KUKA KRL program: Gripper_check.src, Gripper_check.dat

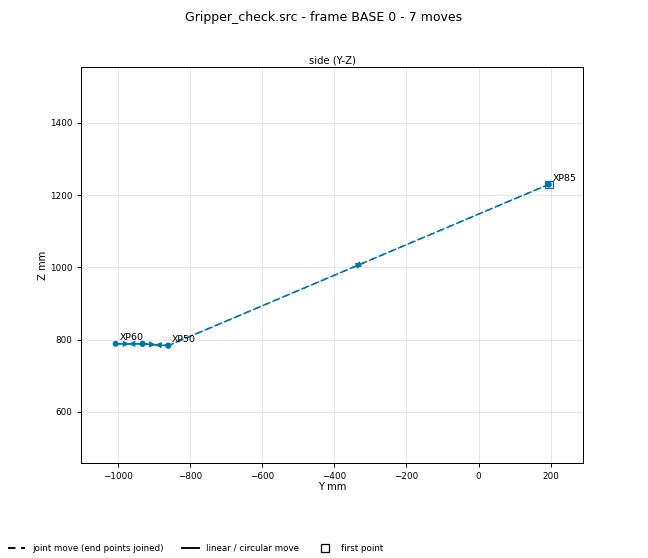
[picture p0: tool path of Gripper_check.src in frame BASE 0, 7 of 9 moves have a stored position in this frame; points joined in program order, loops and branches not executed]
--- Gripper_check.src ---
&ACCESS RVP
&REL 175
&PARAM EDITMASK = *
&PARAM TEMPLATE = C:\KRC\Roboter\Template\vorgabe
&PARAM DISKPATH = KRC:\R1\Program\Sevice Programs
DEF Gripper_check( )
;FOLD INI;%{PE}
  ;FOLD BASISTECH INI
    GLOBAL INTERRUPT DECL 3 WHEN $STOPMESS==TRUE DO IR_STOPM ( )
    INTERRUPT ON 3
    BAS (#INITMOV,0 )
  ;ENDFOLD (BASISTECH INI)
;FOLD SPOTTECH INI
USERSPOT(#INIT)
;ENDFOLD (SPOTTECH INI)
;FOLD GRIPPERTECH INI
USER_GRP(0,DUMMY,DUMMY,GDEFAULT)
;ENDFOLD (GRIPPERTECH INI)
  ;FOLD USER INI
    ;Make your modifications here

  ;ENDFOLD (USER INI)
;ENDFOLD (INI)

;FOLD PTP HOME  Vel= 100 % DEFAULT;%{PE}%MKUKATPBASIS,%CMOVE,%VPTP,%P 1:PTP, 2:HOME, 3:, 5:100, 7:DEFAULT
$BWDSTART = FALSE
PDAT_ACT=PDEFAULT
FDAT_ACT=FHOME
BAS (#PTP_PARAMS,100 )
$H_POS=XHOME
PTP  XHOME
;ENDFOLD

;FOLD PTP P85 Vel=100 % H Tool[5] Base[0];%{PE}%R 8.3.48,%MKUKATPBASIS,%CMOVE,%VPTP,%P 1:PTP, 2:P85, 3:, 5:100, 7:H
$BWDSTART=FALSE
PDAT_ACT=PH
FDAT_ACT=FP85
BAS(#PTP_PARAMS,100)
PTP XP85
;ENDFOLD
;FOLD PTP P50 Vel=100 % H Tool[5] Base[0];%{PE}%R 8.3.48,%MKUKATPBASIS,%CMOVE,%VPTP,%P 1:PTP, 2:P50, 3:, 5:100, 7:H
$BWDSTART=FALSE
PDAT_ACT=PH
FDAT_ACT=FP50
BAS(#PTP_PARAMS,100)
PTP XP50
;ENDFOLD

;FOLD WAIT FOR ( IN 246 'Grps: bat reposo' ) CONT;%{PE}%R 8.3.48 %MKUKATPBASIS %CEXT_WAIT_FOR %VEXT_WAIT_FOR,%P 2:, 4:, 5:$IN, 6:246, 7:Grps: bat reposo, 9:CONTINUE
CONTINUE
WAIT FOR  ( $IN[246] )
;ENDFOLD
;FOLD WAIT FOR ( IN 248 'Grps: bat reposo' ) CONT;%{PE}%R 8.3.48 %MKUKATPBASIS %CEXT_WAIT_FOR %VEXT_WAIT_FOR,%P 2:, 4:, 5:$IN, 6:248, 7:Grps: bat reposo, 9:CONTINUE
CONTINUE
WAIT FOR  ( $IN[248] )
;ENDFOLD

;FOLD LIN P52 Vel=0.1 m/s M Tool[5] Base[0];%{PE}%R 8.3.48,%MKUKATPBASIS,%CMOVE,%VLIN,%P 1:LIN, 2:P52, 3:, 5:0.1, 7:M
$BWDSTART=FALSE
LDAT_ACT=LM
FDAT_ACT=FP52
BAS(#CP_PARAMS,0.1)
LIN XP52
;ENDFOLD

;Pos Galga
;FOLD LIN P60 Vel=0.01 m/s L Tool[5] Base[0];%{PE}%R 8.3.48,%MKUKATPBASIS,%CMOVE,%VLIN,%P 1:LIN, 2:P60, 3:, 5:0.01, 7:L
$BWDSTART=FALSE
LDAT_ACT=LL
FDAT_ACT=FP60
BAS(#CP_PARAMS,0.01)
LIN XP60
;ENDFOLD
HALT

;Cierra pinchos
;FOLD OUT 243 'cil bat reposo' State=FALSE ;%{PE}%R 8.3.48,%MKUKATPBASIS,%COUT,%VOUTX,%P 2:243, 3:cil bat reposo, 5:FALSE, 6:
$OUT[243]=FALSE
;ENDFOLD
;FOLD OUT 244 'cil bat activo' State=TRUE ;%{PE}%R 8.3.48,%MKUKATPBASIS,%COUT,%VOUTX,%P 2:244, 3:cil bat activo, 5:TRUE, 6:
$OUT[244]=TRUE
;ENDFOLD
;FOLD WAIT FOR ( IN 245 'Grps: bat activo' );%{PE}%R 8.3.48 %MKUKATPBASIS %CEXT_WAIT_FOR %VEXT_WAIT_FOR,%P 2:, 4:, 5:$IN, 6:245, 7:Grps: bat activo, 9:
WAIT FOR  ( $IN[245] )
;ENDFOLD
;FOLD WAIT FOR ( IN 247 'Grps: baterias activo' );%{PE}%R 8.3.48 %MKUKATPBASIS %CEXT_WAIT_FOR %VEXT_WAIT_FOR,%P 2:, 4:, 5:$IN, 6:247, 7:Grps: baterias activo, 9:
WAIT FOR  ( $IN[247] )
;ENDFOLD
HALT

;aBRE pinchos
;FOLD OUT 244 'cil bat activo' State=FALSE ;%{PE}%R 8.3.48,%MKUKATPBASIS,%COUT,%VOUTX,%P 2:244, 3:cil bat activo, 5:FALSE, 6:
$OUT[244]=FALSE
;ENDFOLD
;FOLD OUT 243 'cil bat reposo' State=TRUE ;%{PE}%R 8.3.48,%MKUKATPBASIS,%COUT,%VOUTX,%P 2:243, 3:cil bat reposo, 5:TRUE, 6:
$OUT[243]=TRUE
;ENDFOLD
;FOLD WAIT FOR ( IN 246 'Grps: bat reposo' AND IN 248 'Grps: bat reposo' );%{PE}%R 8.3.48 %MKUKATPBASIS %CEXT_WAIT_FOR %VEXT_WAIT_FOR,%P 2:, 4:, 5:$IN, 6:246, 7:Grps: bat reposo, 8:AND, 9:, 10:$IN, 11:248, 12:Grps: bat reposo, 14:
WAIT FOR  ( $IN[246] AND $IN[248] )
;ENDFOLD
;FOLD WAIT Time=1 sec;%{PE}%R 8.3.48,%MKUKATPBASIS,%CWAIT,%VWAIT,%P 3:1
WAIT SEC 1
;ENDFOLD

;Retirada
;FOLD LIN P55 CONT Vel=2 m/s M Tool[5] Base[0];%{PE}%R 8.3.48,%MKUKATPBASIS,%CMOVE,%VLIN,%P 1:LIN, 2:P55, 3:C_DIS C_DIS, 5:2, 7:M
$BWDSTART=FALSE
LDAT_ACT=LM
FDAT_ACT=FP55
BAS(#CP_PARAMS,2)
LIN XP55 C_DIS C_DIS
;ENDFOLD
;FOLD PTP P54 Vel=100 % H Tool[5] Base[0];%{PE}%R 8.3.48,%MKUKATPBASIS,%CMOVE,%VPTP,%P 1:PTP, 2:P54, 3:, 5:100, 7:H
$BWDSTART=FALSE
PDAT_ACT=PH
FDAT_ACT=FP54
BAS(#PTP_PARAMS,100)
PTP XP54
;ENDFOLD
;FOLD PTP P53 Vel=100 % H Tool[5] Base[0];%{PE}%R 8.3.48,%MKUKATPBASIS,%CMOVE,%VPTP,%P 1:PTP, 2:P53, 3:, 5:100, 7:H
$BWDSTART=FALSE
PDAT_ACT=PH
FDAT_ACT=FP53
BAS(#PTP_PARAMS,100)
PTP XP53
;ENDFOLD
HALT

;FOLD PTP HOME  Vel= 100 % DEFAULT;%{PE}%MKUKATPBASIS,%CMOVE,%VPTP,%P 1:PTP, 2:HOME, 3:, 5:100, 7:DEFAULT
$BWDSTART = FALSE
PDAT_ACT=PDEFAULT
FDAT_ACT=FHOME
BAS (#PTP_PARAMS,100 )
$H_POS=XHOME
PTP  XHOME
;ENDFOLD
END

--- Gripper_check.dat ---
&ACCESS RVP
&REL 175
&PARAM EDITMASK = *
&PARAM TEMPLATE = C:\KRC\Roboter\Template\vorgabe
&PARAM DISKPATH = KRC:\R1\Program\Sevice Programs
DEFDAT  Gripper_check
;FOLD EXTERNAL DECLARATIONS;%{PE}%MKUKATPBASIS,%CEXT,%VCOMMON,%P
;FOLD GRIPPERTECH EXT
EXT  H50 (INT  :IN,INT  :IN,INT  :IN,GRP_TYP  :IN )
;ENDFOLD (GRIPPERTECH EXT)
;FOLD SPOTTECH EXT
EXT  USERSPOT (S_COMMAND  :IN,SPOT_TYPE  :IN )
;ENDFOLD (SPOTTECH EXT)
;FOLD BASISTECH EXT;%{PE}%MKUKATPBASIS,%CEXT,%VEXT,%P
EXT  BAS (BAS_COMMAND  :IN,REAL  :IN )
DECL INT SUCCESS
;ENDFOLD (BASISTECH EXT)
;FOLD USER EXT;%{E}%MKUKATPUSER,%CEXT,%VEXT,%P
;Make your modifications here

;ENDFOLD (USER EXT)
;ENDFOLD (EXTERNAL DECLARATIONS)
DECL BASIS_SUGG_T LAST_BASIS={POINT1[] "P60b                    ",POINT2[] "P60b                    ",CP_PARAMS[] "M                       ",PTP_PARAMS[] "H                       ",CONT[] "                        ",CP_VEL[] "2                       ",PTP_VEL[] "100                     ",SYNC_PARAMS[] "SYNCDAT                 ",SPL_NAME[] "S0                      ",A_PARAMS[] "ADAT0                   "}
DECL E6POS XP50={X 952.374695,Y -860.111694,Z 783.046143,A 80.5366592,B 88.5556259,C 169.570068,S 6,T 26,E1 0.0,E2 0.0,E3 0.0,E4 0.0,E5 0.0,E6 0.0}
DECL FDAT FP50={TOOL_NO 5,BASE_NO 0,IPO_FRAME #BASE,POINT2[] " ",TQ_STATE FALSE}
DECL PDAT PH={VEL 100.000,ACC 100.000,APO_DIST 100.000,APO_MODE #CDIS,GEAR_JERK 50.0000,EXAX_IGN 0}
DECL E6POS XP60={X 952.955505,Y -1005.88715,Z 788.139,A 20.0385742,B 89.1085663,C 109.304688,S 6,T 26,E1 0.0,E2 0.0,E3 0.0,E4 0.0,E5 0.0,E6 0.0}
DECL FDAT FP60={TOOL_NO 5,BASE_NO 0,IPO_FRAME #BASE,POINT2[] " ",TQ_STATE FALSE}
DECL LDAT LL={VEL 2.00000,ACC 25.0000,APO_DIST 100.000,APO_FAC 50.0000,AXIS_VEL 100.000,AXIS_ACC 100.000,ORI_TYP #VAR,CIRC_TYP #BASE,JERK_FAC 50.0000,GEAR_JERK 50.0000,EXAX_IGN 0}
DECL E6POS XP51={X 1024.76611,Y -1067.43542,Z 519.066956,A 55.3303528,B 87.7738342,C 145.849503,S 6,T 26,E1 0.0,E2 0.0,E3 0.0,E4 0.0,E5 0.0,E6 0.0}
DECL FDAT FP51={TOOL_NO 5,BASE_NO 0,IPO_FRAME #BASE,POINT2[] " ",TQ_STATE FALSE}
DECL E6POS XP70={X 1027.60229,Y -977.170227,Z 520.707,A 88.3586,B 88.2946472,C 177.924576,S 6,T 26,E1 0.0,E2 0.0,E3 0.0,E4 0.0,E5 0.0,E6 0.0}
DECL FDAT FP70={TOOL_NO 5,BASE_NO 0,IPO_FRAME #BASE,POINT2[] " ",TQ_STATE FALSE}
DECL E6POS XP52={X 952.798523,Y -931.386414,Z 788.051941,A 20.3578415,B 89.1093369,C 109.624481,S 6,T 26,E1 0.0,E2 0.0,E3 0.0,E4 0.0,E5 0.0,E6 0.0}
DECL FDAT FP52={TOOL_NO 5,BASE_NO 0,IPO_FRAME #BASE,POINT2[] " ",TQ_STATE FALSE}
DECL LDAT LM={VEL 2.00000,ACC 25.0000,APO_DIST 100.000,APO_FAC 50.0000,AXIS_VEL 100.000,AXIS_ACC 100.000,ORI_TYP #VAR,CIRC_TYP #BASE,JERK_FAC 50.0000,GEAR_JERK 50.0000,EXAX_IGN 0}
DECL E6POS XP53={X 938.561218,Y 193.717773,Z 1229.66455,A 174.754501,B 24.9198875,C -153.479370,S 6,T 27,E1 0.0,E2 0.0,E3 0.0,E4 0.0,E5 0.0,E6 0.0}
DECL FDAT FP53={TOOL_NO 5,BASE_NO 0,IPO_FRAME #BASE,POINT2[] " ",TQ_STATE FALSE}
DECL E6POS XP54={X 952.374695,Y -860.111694,Z 783.046143,A 80.5366592,B 88.5556259,C 169.570068,S 6,T 26,E1 0.0,E2 0.0,E3 0.0,E4 0.0,E5 0.0,E6 0.0}
DECL FDAT FP54={TOOL_NO 5,BASE_NO 0,IPO_FRAME #BASE,POINT2[] " ",TQ_STATE FALSE}
DECL E6POS XP55={X 952.798523,Y -931.386414,Z 788.051941,A 20.3578415,B 89.1093369,C 109.624481,S 6,T 26,E1 0.0,E2 0.0,E3 0.0,E4 0.0,E5 0.0,E6 0.0}
DECL FDAT FP55={TOOL_NO 5,BASE_NO 0,IPO_FRAME #BASE,POINT2[] " ",TQ_STATE FALSE}
DECL E6POS XP56={X 1023.94318,Y -901.988892,Z 779.185486,A 84.6670,B 88.5756149,C 177.274,S 6,T 26,E1 0.0,E2 0.0,E3 0.0,E4 0.0,E5 0.0,E6 0.0}
DECL FDAT FP56={TOOL_NO 5,BASE_NO 0,IPO_FRAME #BASE,POINT2[] " ",TQ_STATE FALSE}
DECL E6POS XP57={X 1023.94318,Y -901.988892,Z 779.185486,A 84.6670,B 88.5756149,C 177.274,S 6,T 26,E1 0.0,E2 0.0,E3 0.0,E4 0.0,E5 0.0,E6 0.0}
DECL FDAT FP57={TOOL_NO 5,BASE_NO 0,IPO_FRAME #BASE,POINT2[] " ",TQ_STATE FALSE}
DECL E6POS XP58={X 1023.94318,Y -901.988892,Z 779.185486,A 84.6670,B 88.5756149,C 177.274,S 6,T 26,E1 0.0,E2 0.0,E3 0.0,E4 0.0,E5 0.0,E6 0.0}
DECL FDAT FP58={TOOL_NO 5,BASE_NO 0,IPO_FRAME #BASE,POINT2[] " ",TQ_STATE FALSE}
DECL E6POS XP59={X 1023.94318,Y -901.988892,Z 779.185486,A 84.6670,B 88.5756149,C 177.274,S 6,T 26,E1 0.0,E2 0.0,E3 0.0,E4 0.0,E5 0.0,E6 0.0}
DECL FDAT FP59={TOOL_NO 5,BASE_NO 0,IPO_FRAME #BASE,POINT2[] " ",TQ_STATE FALSE}
DECL E6POS XP61={X 1023.94318,Y -901.988892,Z 779.185486,A 84.6670,B 88.5756149,C 177.274,S 6,T 26,E1 0.0,E2 0.0,E3 0.0,E4 0.0,E5 0.0,E6 0.0}
DECL FDAT FP61={TOOL_NO 5,BASE_NO 0,IPO_FRAME #BASE,POINT2[] " ",TQ_STATE FALSE}
DECL E6POS XP62={X 1023.94318,Y -901.988892,Z 779.185486,A 84.6670,B 88.5756149,C 177.274,S 6,T 26,E1 0.0,E2 0.0,E3 0.0,E4 0.0,E5 0.0,E6 0.0}
DECL FDAT FP62={TOOL_NO 5,BASE_NO 0,IPO_FRAME #BASE,POINT2[] " ",TQ_STATE FALSE}
DECL E6POS XP63={X 1023.94318,Y -901.988892,Z 779.185486,A 84.6670,B 88.5756149,C 177.274,S 6,T 26,E1 0.0,E2 0.0,E3 0.0,E4 0.0,E5 0.0,E6 0.0}
DECL FDAT FP63={TOOL_NO 5,BASE_NO 0,IPO_FRAME #BASE,POINT2[] " ",TQ_STATE FALSE}
DECL E6POS XP64={X 1023.94318,Y -901.988892,Z 779.185486,A 84.6670,B 88.5756149,C 177.274,S 6,T 26,E1 0.0,E2 0.0,E3 0.0,E4 0.0,E5 0.0,E6 0.0}
DECL FDAT FP64={TOOL_NO 5,BASE_NO 0,IPO_FRAME #BASE,POINT2[] " ",TQ_STATE FALSE}
DECL E6POS XP65={X 1023.94318,Y -901.988892,Z 779.185486,A 84.6670,B 88.5756149,C 177.274,S 6,T 26,E1 0.0,E2 0.0,E3 0.0,E4 0.0,E5 0.0,E6 0.0}
DECL FDAT FP65={TOOL_NO 5,BASE_NO 0,IPO_FRAME #BASE,POINT2[] " ",TQ_STATE FALSE}
DECL E6POS XP66={X 1023.94318,Y -901.988892,Z 779.185486,A 84.6670,B 88.5756149,C 177.274,S 6,T 26,E1 0.0,E2 0.0,E3 0.0,E4 0.0,E5 0.0,E6 0.0}
DECL FDAT FP66={TOOL_NO 5,BASE_NO 0,IPO_FRAME #BASE,POINT2[] " ",TQ_STATE FALSE}
DECL E6POS XP67={X 1023.94318,Y -901.988892,Z 779.185486,A 84.6670,B 88.5756149,C 177.274,S 6,T 26,E1 0.0,E2 0.0,E3 0.0,E4 0.0,E5 0.0,E6 0.0}
DECL FDAT FP67={TOOL_NO 5,BASE_NO 0,IPO_FRAME #BASE,POINT2[] " ",TQ_STATE FALSE}
DECL E6POS XP68={X 1023.94318,Y -901.988892,Z 779.185486,A 84.6670,B 88.5756149,C 177.274,S 6,T 26,E1 0.0,E2 0.0,E3 0.0,E4 0.0,E5 0.0,E6 0.0}
DECL FDAT FP68={TOOL_NO 5,BASE_NO 0,IPO_FRAME #BASE,POINT2[] " ",TQ_STATE FALSE}
DECL E6POS XP69={X 1023.94318,Y -901.988892,Z 779.185486,A 84.6670,B 88.5756149,C 177.274,S 6,T 26,E1 0.0,E2 0.0,E3 0.0,E4 0.0,E5 0.0,E6 0.0}
DECL FDAT FP69={TOOL_NO 5,BASE_NO 0,IPO_FRAME #BASE,POINT2[] " ",TQ_STATE FALSE}
DECL E6POS XP71={X 1023.94318,Y -901.988892,Z 779.185486,A 84.6670,B 88.5756149,C 177.274,S 6,T 26,E1 0.0,E2 0.0,E3 0.0,E4 0.0,E5 0.0,E6 0.0}
DECL FDAT FP71={TOOL_NO 5,BASE_NO 0,IPO_FRAME #BASE,POINT2[] " ",TQ_STATE FALSE}
DECL E6POS XP72={X 1023.94318,Y -901.988892,Z 779.185486,A 84.6670,B 88.5756149,C 177.274,S 6,T 26,E1 0.0,E2 0.0,E3 0.0,E4 0.0,E5 0.0,E6 0.0}
DECL FDAT FP72={TOOL_NO 5,BASE_NO 0,IPO_FRAME #BASE,POINT2[] " ",TQ_STATE FALSE}
DECL E6POS XP73={X 1023.94318,Y -901.988892,Z 779.185486,A 84.6670,B 88.5756149,C 177.274,S 6,T 26,E1 0.0,E2 0.0,E3 0.0,E4 0.0,E5 0.0,E6 0.0}
DECL FDAT FP73={TOOL_NO 5,BASE_NO 0,IPO_FRAME #BASE,POINT2[] " ",TQ_STATE FALSE}
DECL E6POS XP74={X 1023.94318,Y -901.988892,Z 779.185486,A 84.6670,B 88.5756149,C 177.274,S 6,T 26,E1 0.0,E2 0.0,E3 0.0,E4 0.0,E5 0.0,E6 0.0}
DECL FDAT FP74={TOOL_NO 5,BASE_NO 0,IPO_FRAME #BASE,POINT2[] " ",TQ_STATE FALSE}
DECL E6POS XP75={X 1023.94318,Y -901.988892,Z 779.185425,A 84.6671295,B 88.5756149,C 177.274139,S 6,T 26,E1 0.0,E2 0.0,E3 0.0,E4 0.0,E5 0.0,E6 0.0}
DECL FDAT FP75={TOOL_NO 5,BASE_NO 0,IPO_FRAME #BASE,POINT2[] " ",TQ_STATE FALSE}
DECL E6POS XP76={X 1023.94318,Y -901.988892,Z 779.185425,A 84.6671295,B 88.5756149,C 177.274139,S 6,T 26,E1 0.0,E2 0.0,E3 0.0,E4 0.0,E5 0.0,E6 0.0}
DECL FDAT FP76={TOOL_NO 5,BASE_NO 0,IPO_FRAME #BASE,POINT2[] " ",TQ_STATE FALSE}
DECL E6POS XP77={X 1023.94318,Y -901.988892,Z 779.185425,A 84.6671295,B 88.5756149,C 177.274139,S 6,T 26,E1 0.0,E2 0.0,E3 0.0,E4 0.0,E5 0.0,E6 0.0}
DECL FDAT FP77={TOOL_NO 5,BASE_NO 0,IPO_FRAME #BASE,POINT2[] " ",TQ_STATE FALSE}
DECL E6POS XP78={X 1023.94318,Y -901.988892,Z 779.185486,A 84.6670,B 88.5756149,C 177.274,S 6,T 26,E1 0.0,E2 0.0,E3 0.0,E4 0.0,E5 0.0,E6 0.0}
DECL FDAT FP78={TOOL_NO 5,BASE_NO 0,IPO_FRAME #BASE,POINT2[] " ",TQ_STATE FALSE}
DECL E6POS XP79={X 1023.94318,Y -901.988892,Z 779.185486,A 84.6670,B 88.5756149,C 177.274,S 6,T 26,E1 0.0,E2 0.0,E3 0.0,E4 0.0,E5 0.0,E6 0.0}
DECL FDAT FP79={TOOL_NO 5,BASE_NO 0,IPO_FRAME #BASE,POINT2[] " ",TQ_STATE FALSE}
DECL E6POS XP80={X 1430.28491,Y -715.362488,Z 925.388062,A 22.5307236,B 4.56420231,C 100.046837,S 6,T 58,E1 0.0,E2 0.0,E3 0.0,E4 0.0,E5 0.0,E6 0.0}
DECL FDAT FP80={TOOL_NO 5,BASE_NO 0,IPO_FRAME #BASE,POINT2[] " ",TQ_STATE FALSE}
DECL E6POS XP81={X 1023.94318,Y -901.988892,Z 779.185486,A 84.6670,B 88.5756149,C 177.274,S 6,T 26,E1 0.0,E2 0.0,E3 0.0,E4 0.0,E5 0.0,E6 0.0}
DECL FDAT FP81={TOOL_NO 5,BASE_NO 0,IPO_FRAME #BASE,POINT2[] " ",TQ_STATE FALSE}
DECL E6POS XP82={X 1023.94318,Y -901.988892,Z 779.185425,A 84.6671295,B 88.5756149,C 177.274139,S 6,T 26,E1 0.0,E2 0.0,E3 0.0,E4 0.0,E5 0.0,E6 0.0}
DECL FDAT FP82={TOOL_NO 5,BASE_NO 0,IPO_FRAME #BASE,POINT2[] " ",TQ_STATE FALSE}
DECL E6POS XP83={X 1023.94318,Y -901.988892,Z 779.185425,A 84.6671295,B 88.5756149,C 177.274139,S 6,T 26,E1 0.0,E2 0.0,E3 0.0,E4 0.0,E5 0.0,E6 0.0}
DECL FDAT FP83={TOOL_NO 5,BASE_NO 0,IPO_FRAME #BASE,POINT2[] " ",TQ_STATE FALSE}
DECL E6POS XP84={X 938.561218,Y 193.717773,Z 1229.66455,A 174.754501,B 24.9198875,C -153.479370,S 6,T 27,E1 0.0,E2 0.0,E3 0.0,E4 0.0,E5 0.0,E6 0.0}
DECL FDAT FP84={TOOL_NO 5,BASE_NO 0,IPO_FRAME #BASE,POINT2[] " ",TQ_STATE FALSE}
DECL E6POS XP85={X 938.561279,Y 193.717789,Z 1229.66455,A 174.754501,B 24.9198856,C -153.479370,S 6,T 27,E1 0.0,E2 0.0,E3 0.0,E4 0.0,E5 0.0,E6 0.0}
DECL FDAT FP85={TOOL_NO 5,BASE_NO 0,IPO_FRAME #BASE,POINT2[] " ",TQ_STATE FALSE}
DECL E6POS XP60B={X 952.955505,Y -1005.88715,Z 788.139,A 20.0385742,B 89.1085663,C 109.304688,S 6,T 26,E1 0.0,E2 0.0,E3 0.0,E4 0.0,E5 0.0,E6 0.0}
DECL FDAT FP60b={TOOL_NO 5,BASE_NO 0,IPO_FRAME #BASE,POINT2[] " ",TQ_STATE FALSE}
ENDDAT
